(* Logix 5000 project; controller Laser_Cutter vendor 1 type 14 code 149 rev 28.11; software revision 28.00 *)

TASK MainTask (continuous, watchdog 500 ms) : MainProgram

MODULES
   Local : vendor 1 type 14 code 149 (Compact 0, rev 28.11)
      DI1 : 1769-IQ16 (Compact 2, rev 1.1, Input RPI 20 ms)
      Discrete_IO : Embedded (Compact 1, rev 3.1, Output RPI 20 ms)
      ASCII_Comms_Modual : vendor 1 type 109 code 66 (Compact 3, rev 2.1, Output RPI 2 ms)   // Modual for serial communication with the laser controller
      MURR_IMPACT_IO_1 : vendor 640 type 7 code 55085 (Ethernet 192.168.1.40, rev 1.1, StandardDataDriven RPI 20 ms)
      MURR_IMPACT_IO_2 : vendor 640 type 7 code 55085 (Ethernet 192.168.1.41, rev 1.1, StandardDataDriven RPI 20 ms)
END_MODULES

TYPE CON_EIP_IN :
STRUCT
   targetPosition : DINT;
   positioningBand : DINT;
   speed : DINT;
   zoneBoundaryPos : DINT;
   zoneBoundaryNeg : DINT;
   acceleration : INT;
   deceleration : INT;
   pressingCurrentLimit : INT;
   loadCurrentThreshold : INT;
   cs1_UNAVAILABLE_0 : BOOL;
   PUSH : BOOL;
   DIR : BOOL;
   INC : BOOL;
   GSL0 : BOOL;
   GSL1 : BOOL;
   MOD0 : BOOL;
   MOD1 : BOOL;
   ASO0 : BOOL;
   ASO1 : BOOL;
   SMOD : BOOL;
   cs1_UNAVAILABLE_11 : BOOL;
   NTC0 : BOOL;
   NTC1 : BOOL;
   cs1_UNAVAILABLE_14 : BOOL;
   cs1_UNAVAILABLE_15 : BOOL;
   DSTR : BOOL;
   HOME : BOOL;
   STP : BOOL;
   RES : BOOL;
   SON : BOOL;
   JISL : BOOL;
   JVEL : BOOL;
   JOG_NEG : BOOL;
   JOG_POS : BOOL;
   cs2_UNAVAILABLE_9 : BOOL;
   cs2_UNAVAILABLE_10 : BOOL;
   cs2_UNAVAILABLE_11 : BOOL;
   cs2_UNAVAILABLE_12 : BOOL;
   cs2_UNAVAILABLE_13 : BOOL;
   RMOD : BOOL;
   BKRL : BOOL;
END_STRUCT
END_TYPE

TYPE CON_EIP_OUT :
STRUCT
   currentPosition : DINT;
   commandCurrent : DINT;
   currentSpeed : DINT;
   alarmCode : INT;
   UNAVAILABLE_14 : SINT;
   UNAVAILABLE_15 : SINT;
   UNAVAILABLE_16 : SINT;
   UNAVAILABLE_17 : SINT;
   UNAVAILABLE_18 : SINT;
   UNAVAILABLE_19 : SINT;
   totalMovingCount : DINT;
   totalMovingDistance : DINT;
   ALML : BOOL;
   ss1_UNAVAILABLE_1 : BOOL;
   ss1_UNAVAILABLE_2 : BOOL;
   ss1_UNAVAILABLE_3 : BOOL;
   ss1_UNAVAILABLE_4 : BOOL;
   ss1_UNAVAILABLE_5 : BOOL;
   ss1_UNAVAILABLE_6 : BOOL;
   ss1_UNAVAILABLE_7 : BOOL;
   ss1_UNAVAILABLE_8 : BOOL;
   ss1_UNAVAILABLE_9 : BOOL;
   ss1_UNAVAILABLE_10 : BOOL;
   ss1_UNAVAILABLE_11 : BOOL;
   ss1_UNAVAILABLE_12 : BOOL;
   ss1_UNAVAILABLE_13 : BOOL;
   ss1_UNAVAILABLE_14 : BOOL;
   ss1_UNAVAILABLE_15 : BOOL;
   PEND : BOOL;
   HEND : BOOL;
   MOVE : BOOL;
   ALM : BOOL;
   SV : BOOL;
   PSFL : BOOL;
   PUSH : BOOL;
   GHMS : BOOL;
   RMDS : BOOL;
   TRQS : BOOL;
   LOAD : BOOL;
   PZONE : BOOL;
   ZONE1 : BOOL;
   ZONE2 : BOOL;
   PWR : BOOL;
   EMGS : BOOL;
END_STRUCT
END_TYPE

TYPE POSITIONS :
STRUCT
   POSITIONS : DINT;
END_STRUCT
END_TYPE

TYPE savedRecipes :   // Array of Saved Recipes from HMI
STRUCT
   programOrder : DINT[20];
   numberOfSteps : DINT;
   numZonesBeforeNextStep : DINT[20];
   numXZones : DINT;
   numYZones : DINT;
   recipeName : STRING;
END_STRUCT
END_TYPE

TYPE savedRecipes111 :   // Array of Recipes Saved from HMI
STRUCT
   A : DINT[20];
   B : DINT[20];
   C : DINT[20];
   D : DINT[20];
   E : DINT[20];
   F : DINT[20];
   G : DINT[20];
   H : DINT[20];
   I : DINT[20];
   J : DINT[20];
   K : DINT[20];
   L : DINT[20];
   M : DINT[20];
   N : DINT[20];
   O : DINT[20];
   P : DINT[20];
   Q : DINT[20];
   R : DINT[20];
   S : DINT[20];
   T : DINT[20];
END_STRUCT
END_TYPE

ADD_ON_INSTRUCTION Value_Within_Tolerance   (* revision 1.0 *)
VAR_OUTPUT
   Within_Tolerance : BOOL; {access Read Only, visible}
END_VAR
VAR_INPUT
   Process_Value : DINT; {required}
   Setpoint_Value : DINT; {required}
   Tolerance : DINT; {required}
END_VAR
VAR
   Hi_Limit : DINT; {access None}
   Lo_Limit : DINT; {access None}
END_VAR

ROUTINE Logic   (* ladder *)
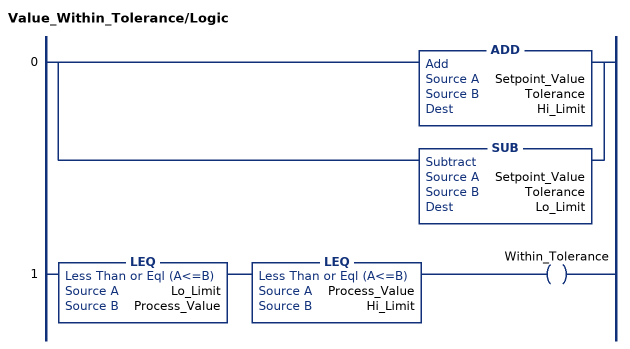
   0: [ADD(Setpoint_Value,Tolerance,Hi_Limit) ,SUB(Setpoint_Value,Tolerance,Lo_Limit) ];
   1: LEQ(Lo_Limit,Process_Value)LEQ(Process_Value,Hi_Limit)OTE(Within_Tolerance);
END_ROUTINE
END_ADD_ON_INSTRUCTION

VAR_GLOBAL   (* controller tags *)
   alarmResetPB : BOOL;   // Global Alarm Reset PB
   audibleAlarm : ALIAS FOR Local:1:O.Data.3;
   bearingConveyorDriveAlarm : ALIAS FOR Local:1:I.Data.6;
   blowOffOn : ALIAS FOR Local:1:O.Data.9;
   boltDriverDown : ALIAS FOR MURR_IMPACT_IO_1:I.Data[1].6;
   boltDriverUp : ALIAS FOR MURR_IMPACT_IO_1:I.Data[1].5;
   boltFeedingBowlOn : ALIAS FOR Local:1:O.Data.7;
   boltFeedingTrackHighLevel : ALIAS FOR MURR_IMPACT_IO_1:I.Data[0].3;
   boltFeedingTrackLowLevel : ALIAS FOR MURR_IMPACT_IO_1:I.Data[0].2;
   boltFeedingTrackOn : ALIAS FOR Local:1:O.Data.8;
   boltPresentAtInfeed : ALIAS FOR MURR_IMPACT_IO_1:I.Data[0].5;
   cameraBadPart : ALIAS FOR Local:1:I.Data.8;
   cameraGoodPart : ALIAS FOR Local:1:I.Data.7;
   cameraOnline : ALIAS FOR Local:1:I.Data.9;
   cameraTrigger : ALIAS FOR Local:1:O.Data.11;
   clampStation2 : ALIAS FOR MURR_IMPACT_IO_1:I.Data[1].7;
   clampStation4 : ALIAS FOR MURR_IMPACT_IO_1:I.Data[2].1;
   clampStation5 : ALIAS FOR MURR_IMPACT_IO_1:I.Data[2].3;
   collarAtStation1 : ALIAS FOR MURR_IMPACT_IO_1:I.Data[0].6;
   collarAtStation2 : ALIAS FOR MURR_IMPACT_IO_1:I.Data[0].7;
   collarAtStation3 : ALIAS FOR MURR_IMPACT_IO_1:I.Data[1].0;
   collarAtStation4 : ALIAS FOR MURR_IMPACT_IO_1:I.Data[1].1;
   collarAtStation5 : ALIAS FOR MURR_IMPACT_IO_1:I.Data[1].2;
   collarFeedingBowlOn : ALIAS FOR Local:1:O.Data.5;
   collarFeedingTrackHighLevel : ALIAS FOR MURR_IMPACT_IO_1:I.Data[0].1;
   collarFeedingTrackLowLevel : ALIAS FOR MURR_IMPACT_IO_1:I.Data[0].0;
   collarFeedingTrackOn : ALIAS FOR Local:1:O.Data.6;
   collarPresentAtInfeed : ALIAS FOR MURR_IMPACT_IO_1:I.Data[0].4;
   currentUser : DINT := 4;   // Access Level of current user
   cycleStartPB : ALIAS FOR Local:1:I.Data.3;
   doorLocksControlRelay : ALIAS FOR Local:1:O.Data.4;
   doorOpenedSafetyRelayStatus : ALIAS FOR Local:1:I.Data.1;
   doorSafetySwitchUnlockSol : ALIAS FOR Local:1:O.Data.10;
   engArrayFullFault : BOOL;
   ESTOP_PB : BOOL;
   eStopSafetyRelayStatus : ALIAS FOR Local:1:I.Data.0;
   greenStatusLight : ALIAS FOR Local:1:O.Data.2;
   keyResetRequired : BOOL;
   leadArrayFullFault : BOOL;
   Local1IData10 : ALIAS FOR Local:1:I.Data.10;
   Local1IData11 : ALIAS FOR Local:1:I.Data.11;
   Local1IData12 : ALIAS FOR Local:1:I.Data.12;
   Local1IData13 : ALIAS FOR Local:1:I.Data.13;
   Local1IData14 : ALIAS FOR Local:1:I.Data.14;
   Local1IData15 : ALIAS FOR Local:1:I.Data.15;
   Local2OData12 : ALIAS FOR Local:1:O.Data.12;
   Local2OData13 : ALIAS FOR Local:1:O.Data.13;
   Local2OData14 : ALIAS FOR Local:1:O.Data.14;
   Local2OData15 : ALIAS FOR Local:1:O.Data.15;
   mainAirOk : ALIAS FOR Local:1:I.Data.2;
   operArrayFullFault : BOOL;
   redStatusLight : ALIAS FOR Local:1:O.Data.0;
   rejectShuttleAtAccept : ALIAS FOR MURR_IMPACT_IO_1:I.Data[2].5;
   rejectShuttleAtReject : ALIAS FOR MURR_IMPACT_IO_1:I.Data[2].6;
   resetPB : ALIAS FOR Local:1:I.Data.5;
   stopPB : ALIAS FOR Local:1:I.Data.4;
   supArrayFullFault : BOOL;
   tapDown : ALIAS FOR MURR_IMPACT_IO_1:I.Data[1].4;
   tapForward : ALIAS FOR MURR_IMPACT_IO_2:O.Data[0].0;
   tapReverse : ALIAS FOR MURR_IMPACT_IO_2:O.Data[0].1;
   tapUp : ALIAS FOR MURR_IMPACT_IO_1:I.Data[1].3;
   TO_DRV1 : CON_EIP_IN := (targetPosition := 12411, positioningBand := 10, speed := 14288, acceleration := 30, deceleration := 30);
   TO_DRV2 : CON_EIP_IN := (targetPosition := 20010, positioningBand := 100, speed := 14288, acceleration := 30, deceleration := 30);
   unclampStation2 : ALIAS FOR MURR_IMPACT_IO_1:I.Data[2].0;
   unclampStation4 : ALIAS FOR MURR_IMPACT_IO_1:I.Data[2].2;
   unclampStation5 : ALIAS FOR MURR_IMPACT_IO_1:I.Data[2].4;
   walkingBeamDown : ALIAS FOR MURR_IMPACT_IO_2:I.Data[0].0;
   walkingBeamLeft : ALIAS FOR MURR_IMPACT_IO_2:I.Data[0].2;
   walkingBeamRight : ALIAS FOR MURR_IMPACT_IO_2:I.Data[0].1;
   walkingBeamUp : ALIAS FOR MURR_IMPACT_IO_1:I.Data[2].7;
   yellowStatusLight : ALIAS FOR Local:1:O.Data.1;
END_VAR

PROGRAM MainProgram   (* main routine MainRoutine *)
VAR
   aAcceptPartSol : BOOL;
   aBlowOffOnSol : BOOL;
   aBlowoffTimer : TIMER := (PRE := 1000);
   aBoltBowlFeedingOn : BOOL;
   aBoltDriverDownSol : BOOL;
   aBoltDriverForward : BOOL;
   aBoltDriverReverse : BOOL;
   aBoltDriverUpSol : BOOL;
   aBoltFeedingTrackOn : BOOL;
   aCameraTrigger : BOOL;
   acceptPartSol : BOOL;
   aClampingStation2Down : BOOL;
   aClampingStation2Up : BOOL;
   aClampingStation4DownSol : BOOL;
   aClampingStation5DownSol : BOOL;
   aClampingStation5UpSol : BOOL;
   aCollarBowlFeedingOn : BOOL;
   aCollarFeedingTrackOn : BOOL;
   aDoorSafetySwitchUnlockSol : BOOL;
   aExhaustStart : BOOL := 1;
   airInitDebounceTimer : TIMER := (PRE := 10000);
   airPressureAlarmTimer : TIMER := (PRE := 4000);
   alarmActive : BOOL;
   alarmActiveOneShot : BOOL;
   alarmActiveOneShotStorage : BOOL;
   alarmMessageBuffer : STRING;
   alarmResetPressed : BOOL;
   alarmResetPressedTmr : TIMER := (PRE := 1000);
   alarmString1 : STRING[35] := ([0] := 'Estop Pressed During Initialization', [1] := 'Door Not Locked During Initialization', [2] := 'Low Air Presure During Initialization', [3] := 'Front Pallet Shotpin Failed to Extend During Initialitzation', [4] := 'Back Pallet Shotpin Failed to Extend During Initialitzation', [5] := 'Estop Pressed During Cycle', [6] := 'Door Opened During Cycle', [7] := 'No Main Air Presure During Cycle', [8] := 'Front Pallet Shotpin Failed to Extend During Cycle', [9] := 'Front Pallet Shotpin Failed to Retract During Cycle', [10] := 'Back Pallet Shotpin Failed to Extend During Cycle', [11] := 'Back Pallet Shotpin Failed to Retract During Cycle', [12] := 'Laser Error', [13] := 'X Axis Failed to Move Home', [14] := 'X Axis Failed to Move to Load', [15] := 'X Axis Failed to Move to Current Zone', [16] := 'X Axis Servo Drive Alarm', [17] := 'X Axis Drive Failed to Enable', [18] := 'X Axis Drive Failed to Disable', [19] := 'Y Axis Failed to Move Home', [20] := 'Y Axis Failed to Move to Load', [21] := 'Y Axis Failed to Move to Current Zone', [22] := 'Y Axis Servo Drive Alarm', [23] := 'Y Axis Drive Failed to Enable', [24] := 'Y Axis Drive Failed to Disable', [25] := 'Laser Timeout Error', [26] := 'External Laser Shutter Failure to Close During Initialization', [27] := 'External Laser Shutter Failure to Close During Cycle', [28] := 'External Laser Shutter Failure to Open During Cycle', [29] := 'Exhaust Arm Not In Position', [30] := 'Low Exhaust Air Flow', [31] := 'User Level Array Full', [32] := 'Low Air Pressure During Cycle', [33] := 'MANUAL MODE ACTIVATED DURING CYCLE');
   alarmString2 : STRING[32];
   alarmStringBuffer : STRING;
   alarmTmr1 : TIMER[32] := ([0].PRE := 100000, [1].PRE := 10000, [2].PRE := 3000, [3].PRE := 3000, [4].PRE := 3000, [5].PRE := 500, [6].PRE := 20000, [7].PRE := 10000, [8].PRE := 10000, [9].PRE := 5000, [10].PRE := 20000, [11].PRE := 10000, [12].PRE := 10000, [13].PRE := 3000, [14].PRE := 20000, [15].PRE := 10000, [16].PRE := 10000, [17].PRE := 3000, [18].PRE := 20000, [19].PRE := 40000, [20].PRE := 10000, [21].PRE := 3000, [22].PRE := 3000, [24].PRE := 500, [25].PRE := 3000, [26].PRE := 3000, [27].PRE := 3000, [28].PRE := 3000, [30].PRE := 3000, [31].PRE := 3000);
   alarmTmr2 : TIMER[32] := ([0].PRE := 3000, [1].PRE := 3000, [2].PRE := 3000, [3].PRE := 3000, [4].PRE := 8000, [5].PRE := 500, [6].PRE := 5000, [7].PRE := 3000, [10].PRE := 3000, [11].PRE := 3000, [13].PRE := 3000, [14].PRE := 3000, [15].PRE := 3000, [17].PRE := 3000, [18].PRE := 3000, [20].PRE := 3000, [21].PRE := 3000, [22].PRE := 3000, [24].PRE := 3000, [25].PRE := 3000, [27].PRE := 3000, [28].PRE := 3000, [30].PRE := 3000);
   aRejectPartSol : BOOL;
   aTapForward : BOOL;
   aTapReverse : BOOL;
   automaticSeqStep : DINT;
   autoMode : BOOL := 1;
   autoModeReady : BOOL := 1;
   aWalkingBeamDownSol : BOOL;
   aWalkingBeamLeftSol : BOOL;
   aWalkingBeamRightSol : BOOL;
   aWalkingBeamUpSol : BOOL;
   blowoffSeqStep : DINT;
   boltBowlFeedingOn : BOOL;
   boltDriverDownDB : TIMER := (PRE := 50);
   boltDriverDownSol : BOOL;
   boltDriverForward : BOOL;
   boltDriverReverse : BOOL;
   boltDriverSeqStep : DINT;
   boltDriverToStartPOS : BOOL;
   boltDriverToStartPOSdb : TIMER := (PRE := 400);
   boltDriverUpDB : TIMER := (PRE := 50);
   boltDriverUpSol : BOOL;
   boltPresentAtInfeedDB : TIMER := (PRE := 50);
   calcZonesDone : BOOL;
   cameraTriggerFlag : BOOL;
   cameraTriggerPulse : TIMER := (PRE := 500);
   clampingStation2Down : BOOL;
   clampingStation2Up : BOOL;
   clampingStation4DownSol : BOOL;
   clampingStation4UpSol : BOOL;
   clampingStation5DownSol : BOOL;
   clampingStation5Sol : BOOL;
   clampStation2DB : TIMER := (PRE := 50);
   clampStation4DB : TIMER := (PRE := 50);
   clampStation5DB : TIMER := (PRE := 50);
   collarAtStation1DB : TIMER := (PRE := 50);
   collarAtStation2DB : TIMER := (PRE := 50);
   collarAtStation3DB : TIMER := (PRE := 50);
   collarAtStation4DB : TIMER := (PRE := 50);
   collarAtStation5DB : TIMER := (PRE := 50);
   collarBowlFeedingOn : BOOL;
   collarFeedingTrackHighLevelDB : TIMER := (PRE := 50);
   collarFeedingTrackLowLevelDB : TIMER := (PRE := 50);
   collarPresentAtInfeedDB : TIMER := (PRE := 50);
   Counter : DINT;
   Counter2 : DINT;
   Counter3 : DINT;
   CYCLE_ALM : DINT;
        .4   // Front Shotpin Failed to Retract During Cycle
        .2   // No Main Air Pressure During Cycle Alarm
        .3   // Front Shotpin Failed to Extend During Cycle
        .1   // Door Opened During Cycle Alarm
        .6   // Back Shotpin Failed to Retract During Cycle
        .5   // Back Shotpin Failed to Extend During Cycle
        .0   // EStop Pressed During Cycle Alarm
        .7   // Laser Error
   CYCLE_ALM_TMR : TIMER[15] := ([3].PRE := 3000, [4].PRE := 3000, [5].PRE := 3000, [6].PRE := 3000, [7].PRE := 3000, [8].PRE := 3000, [9].PRE := 10000, [10].PRE := 250);
   CYCLE_COMPLETE : BOOL;
   CYCLE_IN_PROG : BOOL;
   cycleComplete : BOOL;
   cycleInProgDebounce : TIMER := (PRE := 15000);
   cycleTimeBufferMin : DINT;
   cycleTimeBufferSec : DINT := 2;
   cycleTimer : TIMER := (PRE := 99999999, ACC := 78863958, EN := 1, TT := 1);
   cycleTimerBuffer : DINT;
   doorClosedDebounceTimer : TIMER := (PRE := 50, ACC := 50, EN := 1, DN := 1);
   doorLockAtInitialPosition : BOOL := 1;
   doorLockedDebounceTimer : TIMER := (PRE := 50, ACC := 50, EN := 1, DN := 1);
   doorUnlockedDebounceTimer : TIMER := (PRE := 50);
   empty_string : STRING;
   exeBlowoffSR : BOOL;
   Exec_Bolt_Driver_SR : BOOL;
   Exec_Drive_Bolt : BOOL;
   Exec_Laser_SR : BOOL;
   Exec_Robot_SR : BOOL;
   Exec_Tapping_SR : BOOL;
   execLoadPalletSR : BOOL;
   Execute_BlowoffSR : BOOL;
   Execute_MoveToZoneSR : BOOL;
   Execute_RejectSR : BOOL;
   Execute_VisionInspectionSR : BOOL;
   executeInitializationSequence : BOOL;
   exeCycleStationsSR : BOOL;
   exeInfeedBoltSR : BOOL;
   exeInfeedCollarSR : BOOL;
   exeInspectionSR : BOOL;
   exeRobotSR : BOOL;
   exeScrewBoltSR : BOOL;
   exeTappingSR : BOOL;
   HAND_GREEN_STATUS_LIGHT : BOOL;
   HAND_RED_STATUS_LIGHT : BOOL;
   HAND_YELLOW_STATUS_LIGHT : BOOL;
   HMI_AutoMode_Req : BOOL;
   HMI_ManualMode_Req : BOOL;
   HMI_MESSAGE_NUM : DINT := 16;
   hmiMessageNumber : DINT := 16;
   hmiMessageNumberBuffer : DINT := 16;
   hmiMessageString : STRING := 'READY TO BEGIN CYCLE';
   hmiMessageStringArray : STRING[64] := ([1] := 'ALARM ACTIVE$0D$0APRESS RESET FAULT BUTTON', [2] := 'OFF MODE', [3] := 'MANUAL MODE ACTIVE', [4] := 'EMERGENCY STOP BUTTON PRESSED', [5] := 'RESET OF ESTOP REQUIRED - PUSH RESET BUTTON', [6] := 'SYSTEM INITIALIZATION REQUIRED', [7] := 'INITIALIZATION IN PROGRESS', [8] := 'LASER ERROR - RESET LASER BY TURNING KEY SWITCH OFF AND ON AGAIN', [9] := 'LASER WARNING ACTIVE', [10] := 'DRIVE 1 REQUIRES HOMING', [11] := 'DRIVE 2 REQUIRES HOMING', [12] := 'PALLET NOT PRESENT', [13] := 'CLOSE DOOR AND PRESS POWER ON TO RESET', [14] := 'CYCLE COMPLETE$0D$0AREMOVE PALLET', [15] := 'READY TO LOAD NEW PALLET', [16] := 'READY TO BEGIN CYCLE', [17] := 'AUTOMATIC RUN IN PROGRESS', [18] := 'TEST IN PROGRESS$0D$0APLEASE WAIT', [21] := 'MOVING TO LOAD POSITION FOR END OF RUN$0D$0APLEASE WAIT', [22] := 'REMOVE INSTRUMENT TO COMPLETE RUN', [23] := 'MOVING TO LOAD POSITION TO REPLACE SULU$0D$0APLEASE WAIT', [24] := 'REMOVE INSTRUMENT AND REPLACE SULU', [25] := 'MOVING TO LOAD POSITION$0D$0APLEASE WAIT', [26] := 'MOVING TO 90 DEG MESH LOADING POSITION$0D$0APLEASE WAIT', [27] := 'MOVING TO 65 DEG MESH LOADING POSITION$0D$0APLEASE WAIT', [28] := 'REPLACE 90 DEG MESH AND$0D$0APRESS THE ACKNOWLEDGE BUTTON TO CONFIRM', [29] := 'REPLACE 65 DEG MESH AND$0D$0APRESS THE ACKNOWLEDGE BUTTON TO CONFIRM', [30] := 'ACTIVATE OPTOTOUCH TO MOVE TO LOADING POSITION', [31] := 'ACTIVATE OPTOTOUCH TO MOVE TO LOADING POSITION$0D$0AAFTER THE ALARM', [32] := 'MOVING TO LOADING POSITION$0D$0AAFTER AN ALARM', [33] := 'INSTALL OR RE-POSITION RELIATACK HANDLE NEST', [34] := 'MOVING TO SHORT ABSTACK MESH LOADING POSITION$0D$0APLEASE WAIT', [35] := 'REPLACE SHORT ABSTACK MESH AND$0D$0APRESS THE ACKNOWLEDGE BUTTON TO CONFIRM', [36] := 'MOVING TO LOAD POSITION TO REPLACE INSTRUMENT$0D$0APLEASE WAIT', [37] := 'REMOVE AND REPLACE INSTRUMENT', [50] := 'PRINTING LAST SAMPLE LABELS$0D$0AFOR LABEL CHECKING', [51] := 'PRESS REPRINT ALL LABELS BUTTON', [52] := 'PRINTING SUMMARY LABELS$0D$0APLEASE WAIT', [53] := 'PRESS REPRINT SUMMARY LABELS BUTTON');
   idleTime : TIMER := (PRE := 99999999, ACC := 48278377, EN := 1, TT := 1);
   idleTimeBuffer : DINT;
   idleTimeBufferMin : DINT := 804;
   idleTimeBufferSec : DINT := 38;
   INIT_ALM : DINT;
        .4   // Back Shotpin Failed to Retract During Initialiazation
        .2   // No Main Air Pressure During Initialization Alarm
        .0   // EStop Pressed During Initialization Alarm
        .1   // Door Failed to Lock Durring Initialiaztion
        .3   // Front Shotpin Failed to Retract During Initialiazation
   INIT_ALM_TMR : TIMER[10] := ([3].PRE := 3000, [4].PRE := 3000, [5].PRE := 3000, [6].PRE := 3000);
   INIT_IN_PROG : BOOL;
   INIT_START_PB : BOOL;
   INIT_START_PB_ONS : BOOL;
   initDelayTimer : TIMER := (PRE := 500);
   initHMIMessageDelayTimer : TIMER := (PRE := 500);
   initializationPushbutton : BOOL;
   InitializationRequired : BOOL;
   Initialize_Timer : TIMER := (PRE := 3000, ACC := 3000, EN := 1, DN := 1);
   initSeqStep : DINT;
   initTimeout : TIMER := (PRE := 10000);
   inspectionSeqStep : DINT;
   lampTestActive : BOOL;
   lampTestPB : BOOL;
   lampTestTimer : TIMER := (PRE := 6000);
   laserMessageSeqStep : INT;
   LaserSeqStep : INT;
   leadingZeros : STRING := '000';
   loadPalletSeqStep : INT;
   mAcceptPartPB : BOOL;
   mAcceptPartSol : BOOL;
   manualMode : BOOL;
   maTapReversePB : BOOL;
   mBlowOffOn : BOOL;
   mBlowOffOnSol : BOOL;
   mBlowOffSol : BOOL;
   mBoltBowlFeedingOnPB : BOOL;
   mBoltDriverDownPB : BOOL;
   mBoltDriverDownSol : BOOL;
   mBoltDriverForward : BOOL;
   mBoltDriverForwardPB : BOOL;
   mBoltDriverReverse : BOOL;
   mBoltDriverReversePB : BOOL;
   mBoltDriverUpPB : BOOL;
   mBoltDriverUpSol : BOOL;
   mBoltFeedingTrackOnPB : BOOL;
   mcameraTrigger : BOOL;
   mClampingStation2Down : BOOL;
   mClampingStation2DownSol : BOOL;
   mClampingStation2Up : BOOL;
   mClampingStation2UpPB : BOOL;
   mClampingStation2UpSol : BOOL;
   mClampingStation4DownSol : BOOL;
   mClampingStation4UpPB : BOOL;
   mClampingStation4UpSol : BOOL;
   mClampingStation5DownPB : BOOL;
   mClampingStation5DownSol : BOOL;
   mClampingStation5UpPB : BOOL;
   mClampingStation5UpSol : BOOL;
   mClampStation4DownPB : BOOL;
   mCollarBowlFeedingOnPB : BOOL;
   mCollarFeedingTrackOnPB : BOOL;
   mDoorSafetySwitchUnlockSol : BOOL;
   MoveToZoneSeqStep : INT;
   mRejectPartPB : BOOL;
   mRejectPartSol : BOOL;
   mSecPulseOffTmr1 : TIMER;
   mSecPulseOnTmr1 : TIMER := (EN := 1, TT := 1);
   mTapForward : BOOL;
   mTapForwardPB : BOOL;
   mTapReverse : BOOL;
   mWalkingBeamDownPB : BOOL;
   mWalkingBeamDownSol : BOOL;
   mWalkingBeamLeftPB : BOOL;
   mWalkingBeamLeftSol : BOOL;
   mWalkingBeamRightPB : BOOL;
   mWalkingBeamRightSol : BOOL;
   mWalkingBeamUpPB : BOOL;
   mWalkingBeamUpSol : BOOL;
   n : TIMER := (PRE := 50);
   noAirDurringCycleAlarmTimer : TIMER := (PRE := 3000);
   nulString : STRING;
   oneSecPulseOffTmr : TIMER := (EN := 1, TT := 1);
   oneSecPulseOnTmr : TIMER;
   p2pCycleTime : TIMER := (PRE := 99999999, ACC := 2605);
   p2pCycleTimeBuffer : DINT := 10001;
   p2pCycleTimeBufferSec : DINT := 10;
   palletpresentDebounceTimer : TIMER := (PRE := 50, ACC := 51, EN := 1, DN := 1);
   palletShotpinExtendedBackDebounceTimer : TIMER := (PRE := 50);
   palletShotpinExtendedFrontDebounceTimer : TIMER := (PRE := 50);
   palletShotpinRetractedDebounceTimer : TIMER := (PRE := 50, ACC := 51, EN := 1, DN := 1);
   partsPresentDurringInitialization : BOOL;
   pause : BOOL := 1;
   performOpControl : CONTROL := (LEN := 6);
   performOperation : DINT[1];
   readyToMovePallet : BOOL;
   readyToStartCycle : BOOL;
   rejectPartFlag : BOOL;
   rejectPartSol : BOOL;
   rejectPartSR : DINT[1];
   rejectSeqStep : DINT;
   rejectShuttleAtAcceptDB : TIMER := (PRE := 50);
   rejectShuttleAtRejectDB : TIMER := (PRE := 50);
   remotePVDisplayNum : DINT;
   resetPartCountingValuesHMIPB : BOOL;
   resetPartCountingValuesTimer : TIMER := (PRE := 3000);
   robotAtDropAPR : BOOL;
   robotAtHome : BOOL;
   robotAtPickAPR : BOOL;
   robotFinishedDrop : BOOL;
   robotHasBolt : BOOL;
   robotInMotion : BOOL;
   robotPickBolt : BOOL;
   robotScrewInBolt : BOOL;
   robotSeqStep : DINT;
   runsCompleted : DINT := 100;
   runTime : TIMER := (PRE := 99999999);
   runTimeBuffer : DINT;
   runTimeBufferMin : DINT;
   runTimeBufferSec : DINT;
   sendRobotToDropAPR : BOOL;
   sendRobotToHome : BOOL;
   sendRobotToPick : BOOL;
   serialPortControl : SERIAL_PORT_CONTROL;
   shortDelay : TIMER := (PRE := 50);
   startCycleTimer : BOOL := 1;
   startP2PTimer : BOOL := 1;
   startRobotSequence : BOOL;
   startRunTimer : BOOL;
   stationNumber : CONTROL := (LEN := 6, POS := 5);
   systemInInitializedPosition : BOOL := 1;
   tapDownDB : TIMER := (PRE := 50);
   tapDwellTimer : TIMER := (PRE := 250);
   tapSeqStep : DINT := 40;
   tapUpDB : TIMER := (PRE := 50);
   testInProgress : BOOL;
   testLaserInZonePB : BOOL := 1;
   testLaserInZonePBONs : BOOL;
   testToggle : BOOL;
   testToggle2 : BOOL := 1;
   TMR_PULSE_OFF : TIMER := (PRE := 500);
   TMR_PULSE_ON : TIMER := (PRE := 500, ACC := 296, EN := 1, TT := 1);
   unclampStation2DB : TIMER := (PRE := 50);
   unclampStation4DB : TIMER := (PRE := 50);
   unclampStation5DB : TIMER := (PRE := 50);
   walkingBeamDownDB : TIMER := (PRE := 50, ACC := 51);
   walkingBeamDownSol : BOOL;
   walkingBeamLeftDB : TIMER := (PRE := 50);
   walkingBeamLeftSol : BOOL;
   walkingBeamRightDB : TIMER := (PRE := 50, ACC := 51);
   walkingBeamRightSol : BOOL;
   walkingBeamUpDB : TIMER := (PRE := 50);
   walkingBeamUpSol : BOOL;
END_VAR

ROUTINE Alarms   (* ladder *)
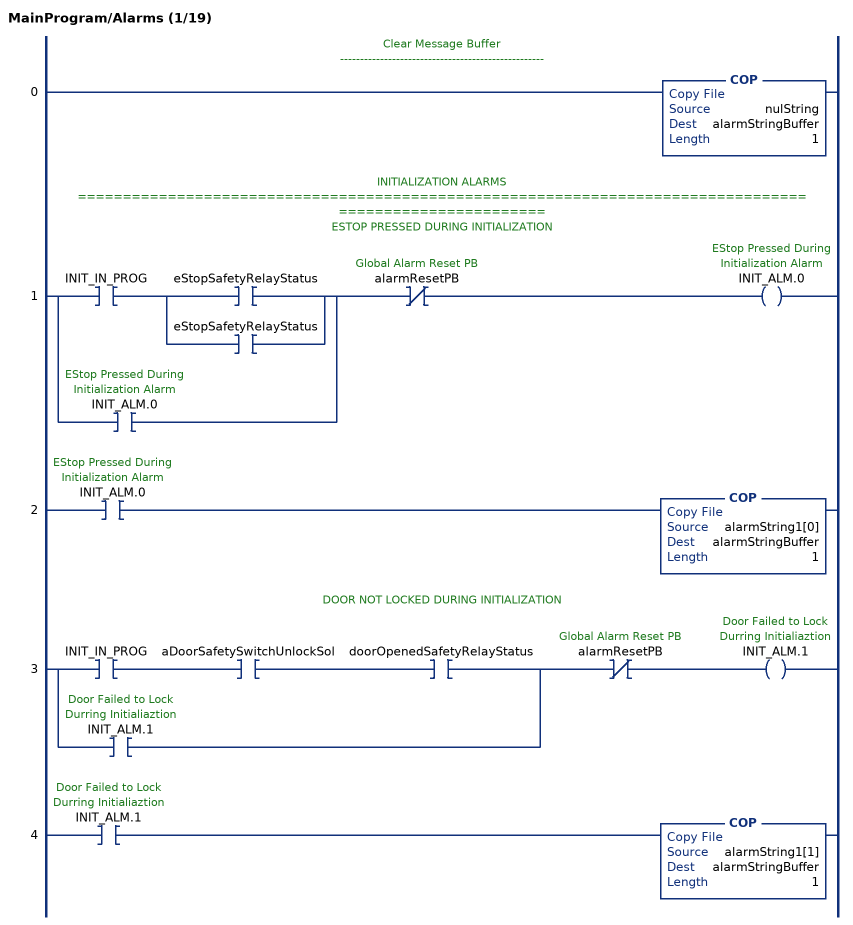
   // Clear Message Buffer
   // ---------------------------------------------------
   0: COP(nulString,alarmStringBuffer,1);
   // INITIALIZATION ALARMS
   // ========================================================================================================
   // ESTOP PRESSED DURING INITIALIZATION
   1: [XIC(INIT_IN_PROG) [XIC(eStopSafetyRelayStatus) ,XIC(eStopSafetyRelayStatus) ] ,XIC(INIT_ALM.0) ]XIO(alarmResetPB)OTE(INIT_ALM.0);
   2: XIC(INIT_ALM.0)COP(alarmString1[0],alarmStringBuffer,1);
   // DOOR NOT LOCKED DURING INITIALIZATION
   3: [XIC(INIT_IN_PROG) XIC(aDoorSafetySwitchUnlockSol) XIC(doorOpenedSafetyRelayStatus) ,XIC(INIT_ALM.1) ]XIO(alarmResetPB)OTE(INIT_ALM.1);
   4: XIC(INIT_ALM.1)COP(alarmString1[1],alarmStringBuffer,1);
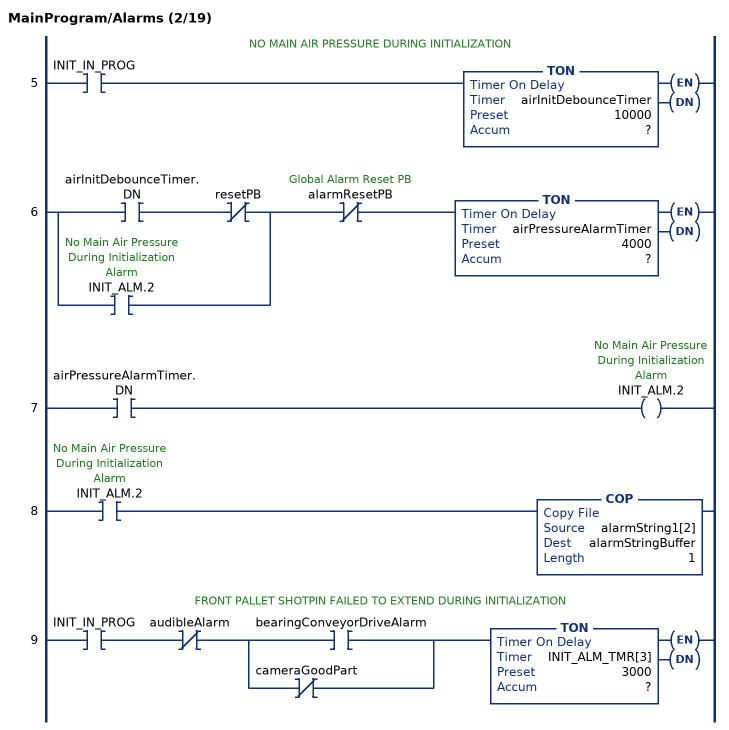
   // NO MAIN AIR PRESSURE DURING INITIALIZATION
   5: XIC(INIT_IN_PROG)TON(airInitDebounceTimer,?,?);
   6: [XIC(airInitDebounceTimer.DN) XIO(resetPB) ,XIC(INIT_ALM.2) ]XIO(alarmResetPB)TON(airPressureAlarmTimer,?,?);
   7: XIC(airPressureAlarmTimer.DN)OTE(INIT_ALM.2);
   8: XIC(INIT_ALM.2)COP(alarmString1[2],alarmStringBuffer,1);
   // FRONT PALLET SHOTPIN FAILED TO EXTEND DURING INITIALIZATION
   9: XIC(INIT_IN_PROG)XIO(audibleAlarm)[XIC(bearingConveyorDriveAlarm) ,XIO(cameraGoodPart) ]TON(INIT_ALM_TMR[3],?,?);
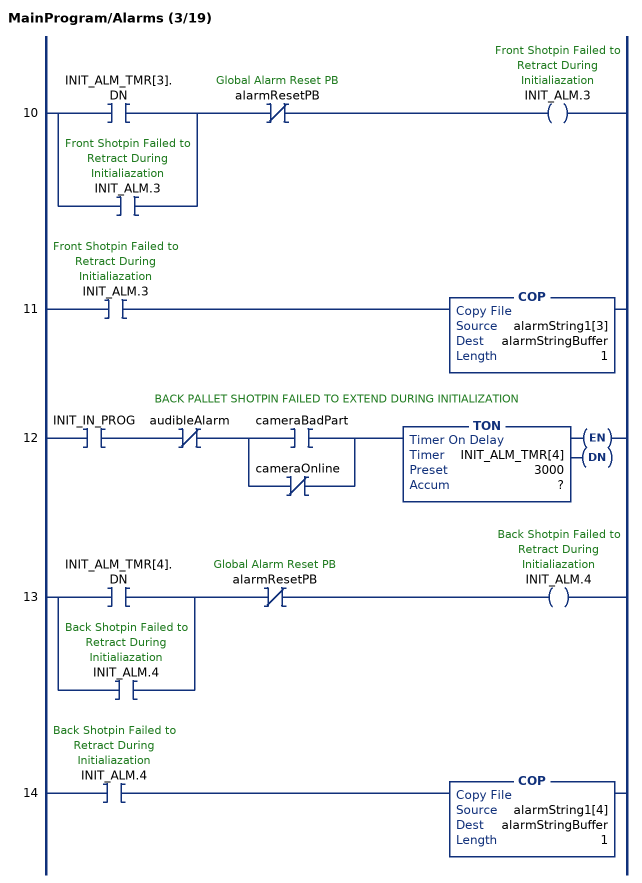
   10: [XIC(INIT_ALM_TMR[3].DN) ,XIC(INIT_ALM.3) ]XIO(alarmResetPB)OTE(INIT_ALM.3);
   11: XIC(INIT_ALM.3)COP(alarmString1[3],alarmStringBuffer,1);
   // BACK PALLET SHOTPIN FAILED TO EXTEND DURING INITIALIZATION
   12: XIC(INIT_IN_PROG)XIO(audibleAlarm)[XIC(cameraBadPart) ,XIO(cameraOnline) ]TON(INIT_ALM_TMR[4],?,?);
   13: [XIC(INIT_ALM_TMR[4].DN) ,XIC(INIT_ALM.4) ]XIO(alarmResetPB)OTE(INIT_ALM.4);
   14: XIC(INIT_ALM.4)COP(alarmString1[4],alarmStringBuffer,1);
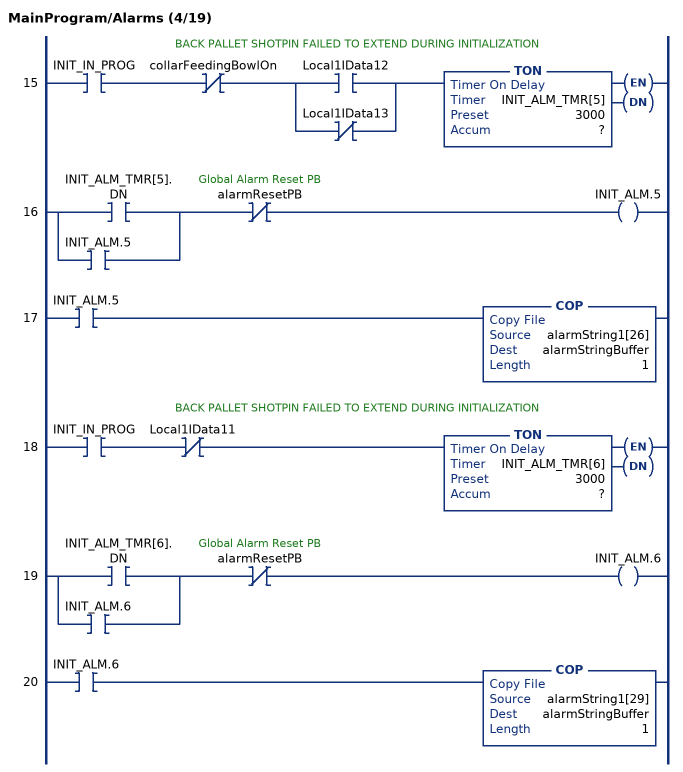
   // BACK PALLET SHOTPIN FAILED TO EXTEND DURING INITIALIZATION
   15: XIC(INIT_IN_PROG)XIO(collarFeedingBowlOn)[XIC(Local1IData12) ,XIO(Local1IData13) ]TON(INIT_ALM_TMR[5],?,?);
   16: [XIC(INIT_ALM_TMR[5].DN) ,XIC(INIT_ALM.5) ]XIO(alarmResetPB)OTE(INIT_ALM.5);
   17: XIC(INIT_ALM.5)COP(alarmString1[26],alarmStringBuffer,1);
   // BACK PALLET SHOTPIN FAILED TO EXTEND DURING INITIALIZATION
   18: XIC(INIT_IN_PROG)XIO(Local1IData11)TON(INIT_ALM_TMR[6],?,?);
   19: [XIC(INIT_ALM_TMR[6].DN) ,XIC(INIT_ALM.6) ]XIO(alarmResetPB)OTE(INIT_ALM.6);
   20: XIC(INIT_ALM.6)COP(alarmString1[29],alarmStringBuffer,1);
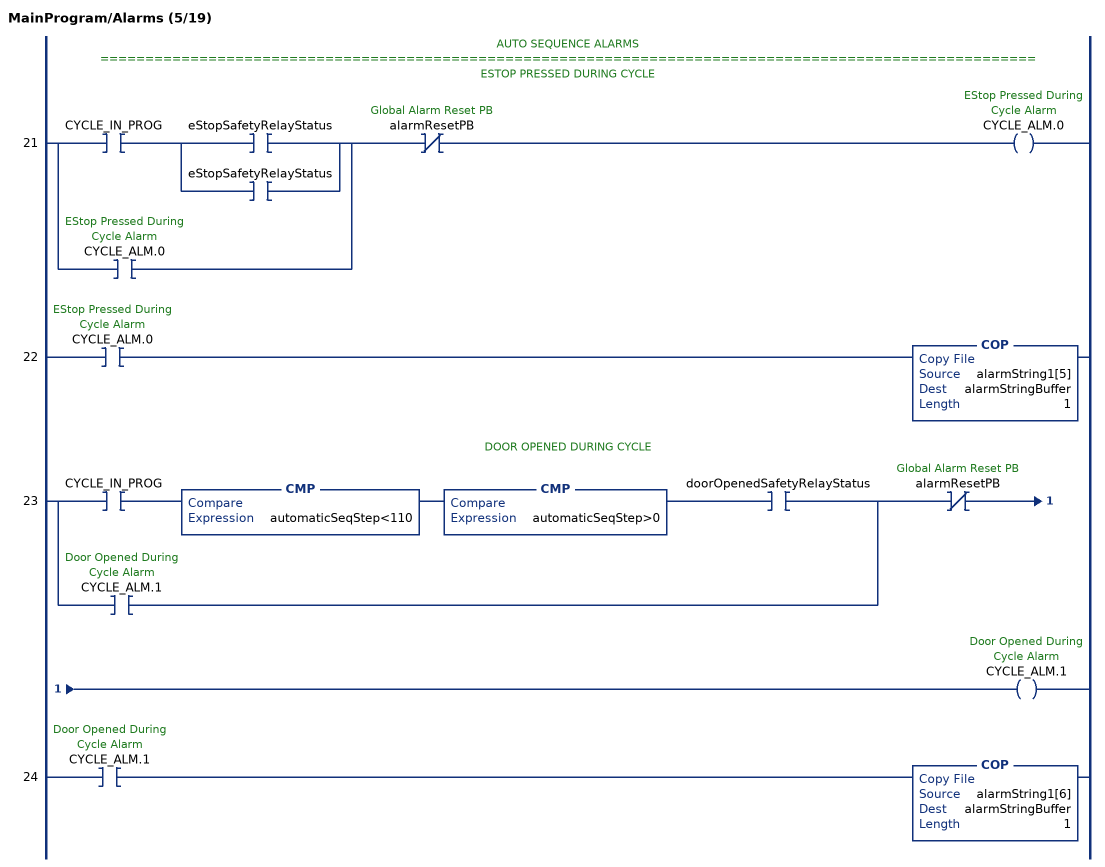
   // AUTO SEQUENCE ALARMS
   // ========================================================================================================
   // ESTOP PRESSED DURING CYCLE
   21: [XIC(CYCLE_IN_PROG) [XIC(eStopSafetyRelayStatus) ,XIC(eStopSafetyRelayStatus) ] ,XIC(CYCLE_ALM.0) ]XIO(alarmResetPB)OTE(CYCLE_ALM.0);
   22: XIC(CYCLE_ALM.0)COP(alarmString1[5],alarmStringBuffer,1);
   // DOOR OPENED DURING CYCLE
   23: [XIC(CYCLE_IN_PROG) CMP(automaticSeqStep<110) CMP(automaticSeqStep>0) XIC(doorOpenedSafetyRelayStatus) ,XIC(CYCLE_ALM.1) ]XIO(alarmResetPB)OTE(CYCLE_ALM.1);
   24: XIC(CYCLE_ALM.1)COP(alarmString1[6],alarmStringBuffer,1);
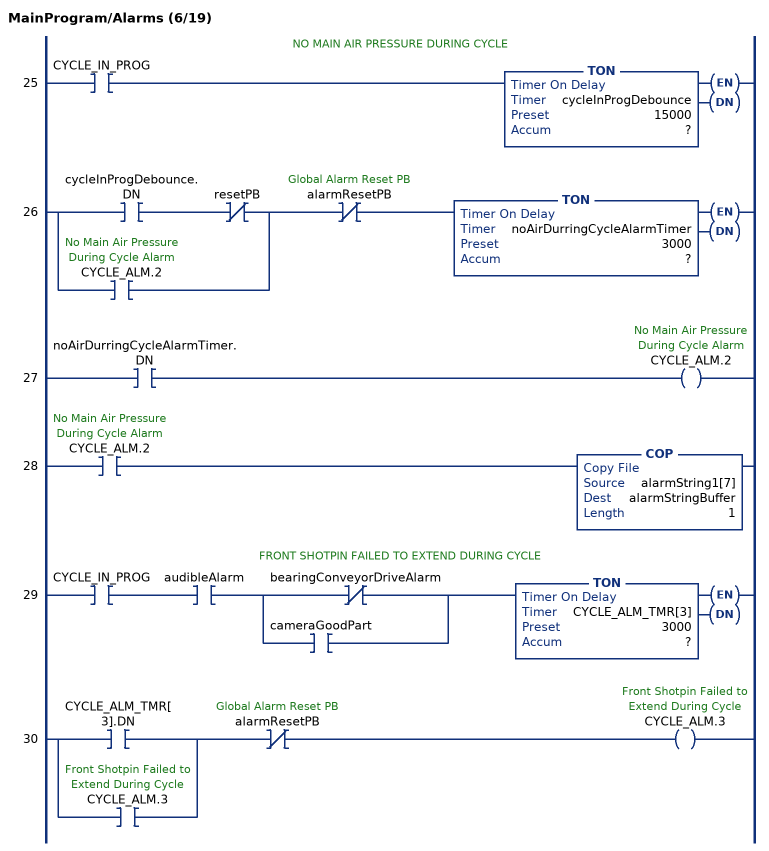
   // NO MAIN AIR PRESSURE DURING CYCLE
   25: XIC(CYCLE_IN_PROG)TON(cycleInProgDebounce,?,?);
   26: [XIC(cycleInProgDebounce.DN) XIO(resetPB) ,XIC(CYCLE_ALM.2) ]XIO(alarmResetPB)TON(noAirDurringCycleAlarmTimer,?,?);
   27: XIC(noAirDurringCycleAlarmTimer.DN)OTE(CYCLE_ALM.2);
   28: XIC(CYCLE_ALM.2)COP(alarmString1[7],alarmStringBuffer,1);
   // FRONT SHOTPIN FAILED TO EXTEND DURING CYCLE
   29: XIC(CYCLE_IN_PROG)XIC(audibleAlarm)[XIO(bearingConveyorDriveAlarm) ,XIC(cameraGoodPart) ]TON(CYCLE_ALM_TMR[3],?,?);
   30: [XIC(CYCLE_ALM_TMR[3].DN) ,XIC(CYCLE_ALM.3) ]XIO(alarmResetPB)OTE(CYCLE_ALM.3);
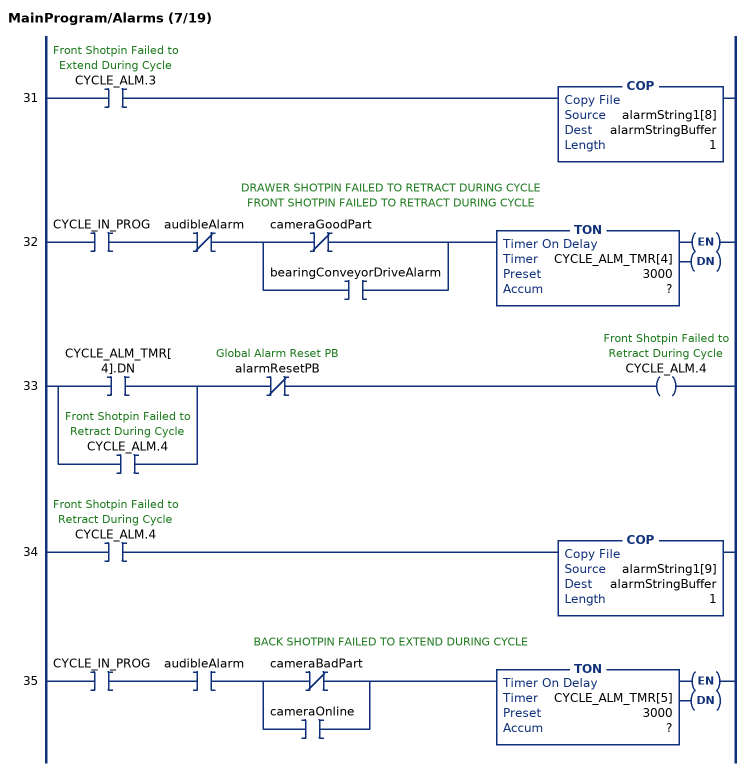
   31: XIC(CYCLE_ALM.3)COP(alarmString1[8],alarmStringBuffer,1);
   // DRAWER SHOTPIN FAILED TO RETRACT DURING CYCLE
   // FRONT SHOTPIN FAILED TO RETRACT DURING CYCLE
   32: XIC(CYCLE_IN_PROG)XIO(audibleAlarm)[XIO(cameraGoodPart) ,XIC(bearingConveyorDriveAlarm) ]TON(CYCLE_ALM_TMR[4],?,?);
   33: [XIC(CYCLE_ALM_TMR[4].DN) ,XIC(CYCLE_ALM.4) ]XIO(alarmResetPB)OTE(CYCLE_ALM.4);
   34: XIC(CYCLE_ALM.4)COP(alarmString1[9],alarmStringBuffer,1);
   // BACK SHOTPIN FAILED TO EXTEND DURING CYCLE
   35: XIC(CYCLE_IN_PROG)XIC(audibleAlarm)[XIO(cameraBadPart) ,XIC(cameraOnline) ]TON(CYCLE_ALM_TMR[5],?,?);
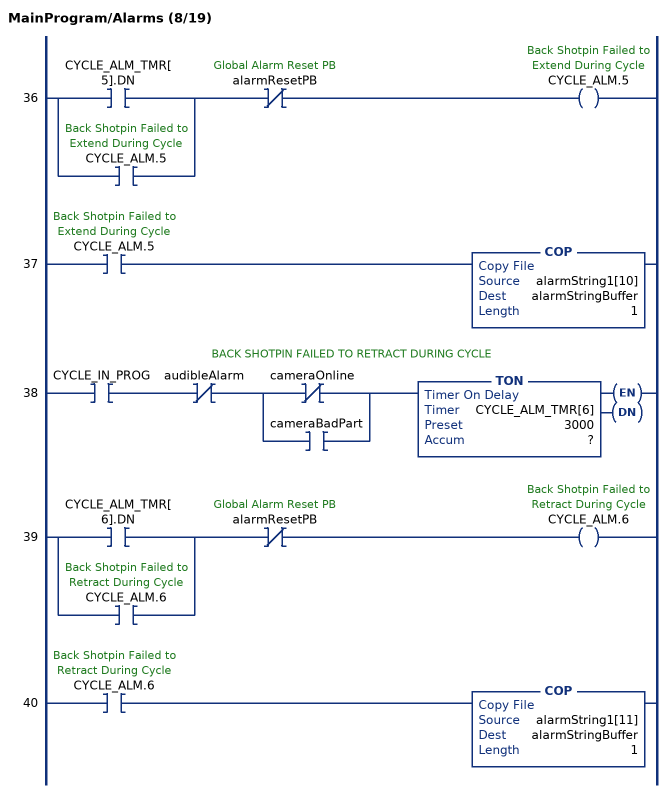
   36: [XIC(CYCLE_ALM_TMR[5].DN) ,XIC(CYCLE_ALM.5) ]XIO(alarmResetPB)OTE(CYCLE_ALM.5);
   37: XIC(CYCLE_ALM.5)COP(alarmString1[10],alarmStringBuffer,1);
   // BACK SHOTPIN FAILED TO RETRACT DURING CYCLE
   38: XIC(CYCLE_IN_PROG)XIO(audibleAlarm)[XIO(cameraOnline) ,XIC(cameraBadPart) ]TON(CYCLE_ALM_TMR[6],?,?);
   39: [XIC(CYCLE_ALM_TMR[6].DN) ,XIC(CYCLE_ALM.6) ]XIO(alarmResetPB)OTE(CYCLE_ALM.6);
   40: XIC(CYCLE_ALM.6)COP(alarmString1[11],alarmStringBuffer,1);
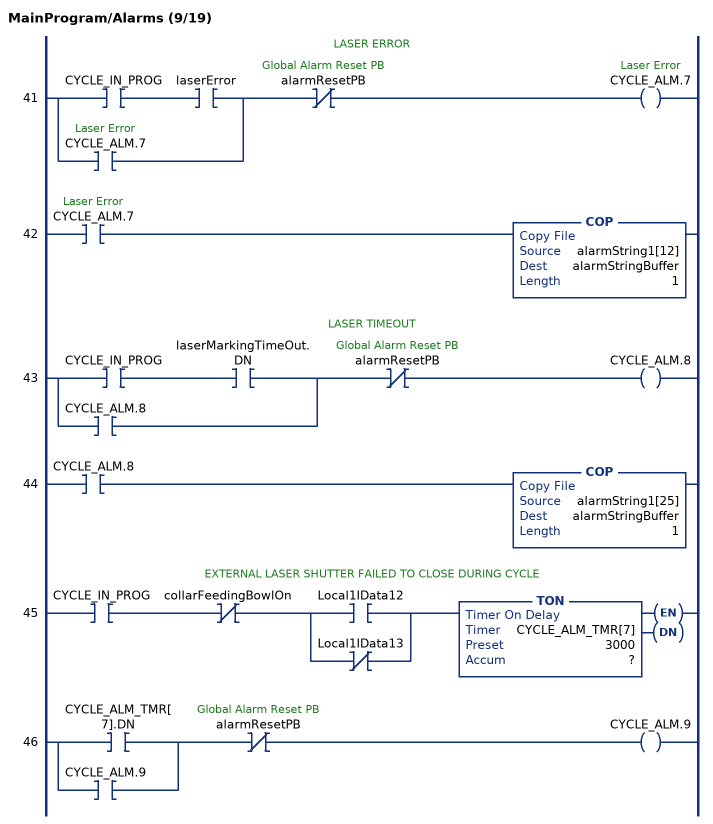
   // LASER ERROR
   41: [XIC(CYCLE_IN_PROG) XIC(laserError) ,XIC(CYCLE_ALM.7) ]XIO(alarmResetPB)OTE(CYCLE_ALM.7);
   42: XIC(CYCLE_ALM.7)COP(alarmString1[12],alarmStringBuffer,1);
   // LASER TIMEOUT
   43: [XIC(CYCLE_IN_PROG) XIC(laserMarkingTimeOut.DN) ,XIC(CYCLE_ALM.8) ]XIO(alarmResetPB)OTE(CYCLE_ALM.8);
   44: XIC(CYCLE_ALM.8)COP(alarmString1[25],alarmStringBuffer,1);
   // EXTERNAL LASER SHUTTER FAILED TO CLOSE DURING CYCLE
   45: XIC(CYCLE_IN_PROG)XIO(collarFeedingBowlOn)[XIC(Local1IData12) ,XIO(Local1IData13) ]TON(CYCLE_ALM_TMR[7],?,?);
   46: [XIC(CYCLE_ALM_TMR[7].DN) ,XIC(CYCLE_ALM.9) ]XIO(alarmResetPB)OTE(CYCLE_ALM.9);
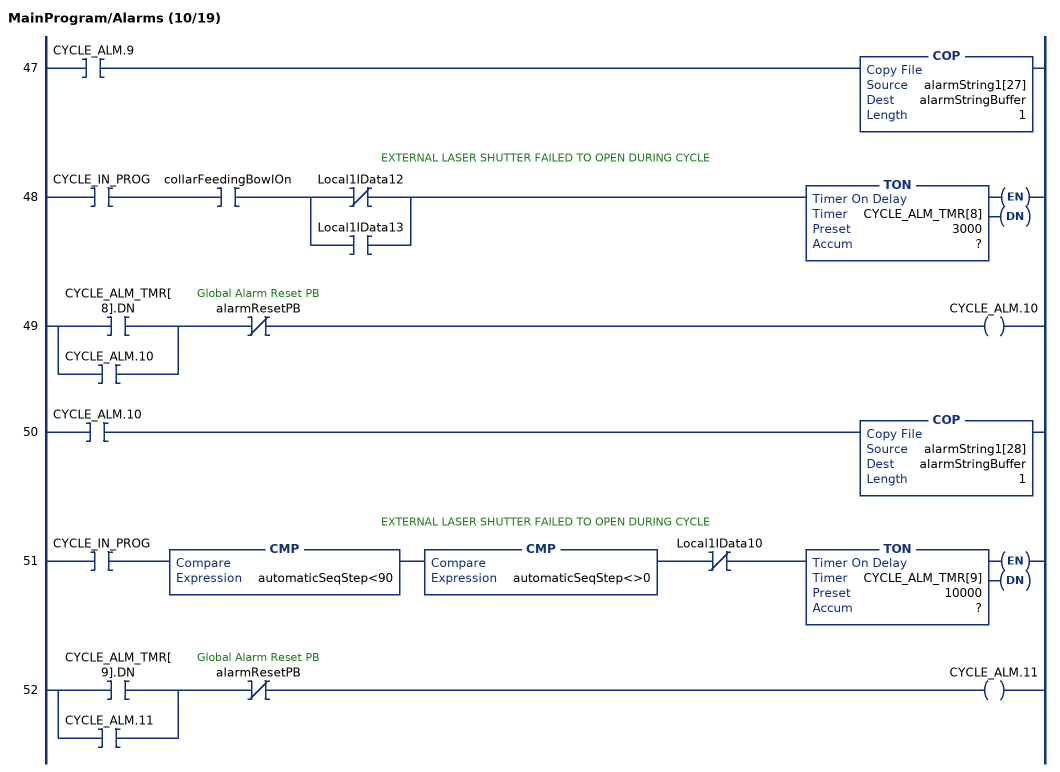
   47: XIC(CYCLE_ALM.9)COP(alarmString1[27],alarmStringBuffer,1);
   // EXTERNAL LASER SHUTTER FAILED TO OPEN DURING CYCLE
   48: XIC(CYCLE_IN_PROG)XIC(collarFeedingBowlOn)[XIO(Local1IData12) ,XIC(Local1IData13) ]TON(CYCLE_ALM_TMR[8],?,?);
   49: [XIC(CYCLE_ALM_TMR[8].DN) ,XIC(CYCLE_ALM.10) ]XIO(alarmResetPB)OTE(CYCLE_ALM.10);
   50: XIC(CYCLE_ALM.10)COP(alarmString1[28],alarmStringBuffer,1);
   // EXTERNAL LASER SHUTTER FAILED TO OPEN DURING CYCLE
   51: XIC(CYCLE_IN_PROG)CMP(automaticSeqStep<90)CMP(automaticSeqStep<>0)XIO(Local1IData10)TON(CYCLE_ALM_TMR[9],?,?);
   52: [XIC(CYCLE_ALM_TMR[9].DN) ,XIC(CYCLE_ALM.11) ]XIO(alarmResetPB)OTE(CYCLE_ALM.11);
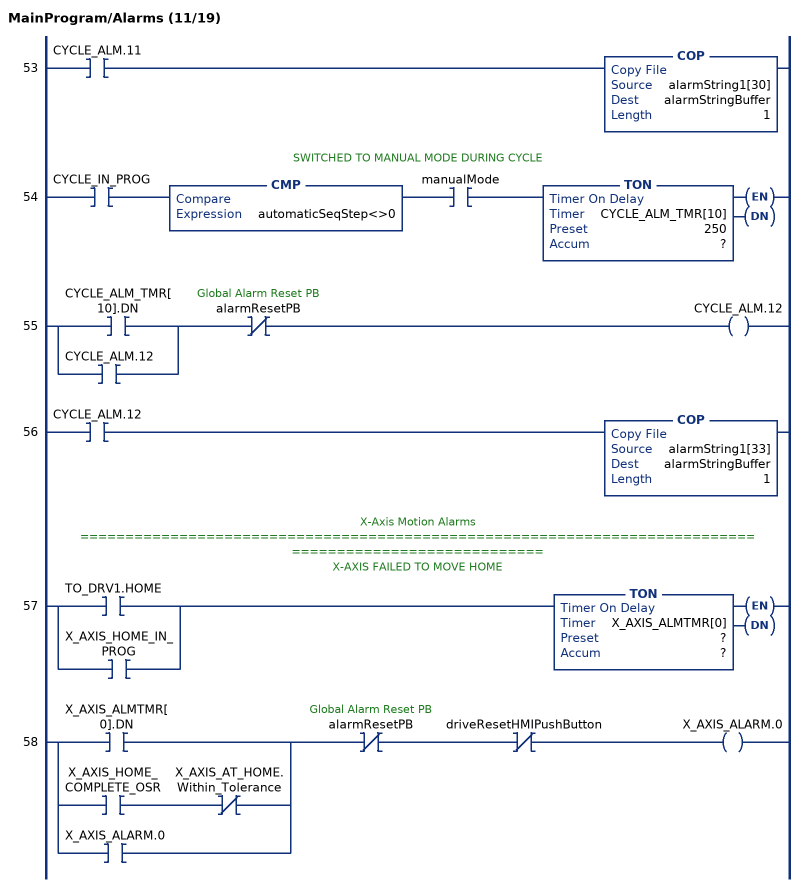
   53: XIC(CYCLE_ALM.11)COP(alarmString1[30],alarmStringBuffer,1);
   // SWITCHED TO MANUAL MODE DURING CYCLE
   54: XIC(CYCLE_IN_PROG)CMP(automaticSeqStep<>0)XIC(manualMode)TON(CYCLE_ALM_TMR[10],?,?);
   55: [XIC(CYCLE_ALM_TMR[10].DN) ,XIC(CYCLE_ALM.12) ]XIO(alarmResetPB)OTE(CYCLE_ALM.12);
   56: XIC(CYCLE_ALM.12)COP(alarmString1[33],alarmStringBuffer,1);
   // X-Axis Motion Alarms
   // =======================================================================================================
   // X-AXIS FAILED TO MOVE HOME
   57: [XIC(TO_DRV1.HOME) ,XIC(X_AXIS_HOME_IN_PROG) ]TON(X_AXIS_ALMTMR[0],?,?);
   58: [XIC(X_AXIS_ALMTMR[0].DN) ,XIC(X_AXIS_HOME_COMPLETE_OSR) XIO(X_AXIS_AT_HOME.Within_Tolerance) ,XIC(X_AXIS_ALARM.0) ]XIO(alarmResetPB)XIO(driveResetHMIPushButton)OTE(X_AXIS_ALARM.0);
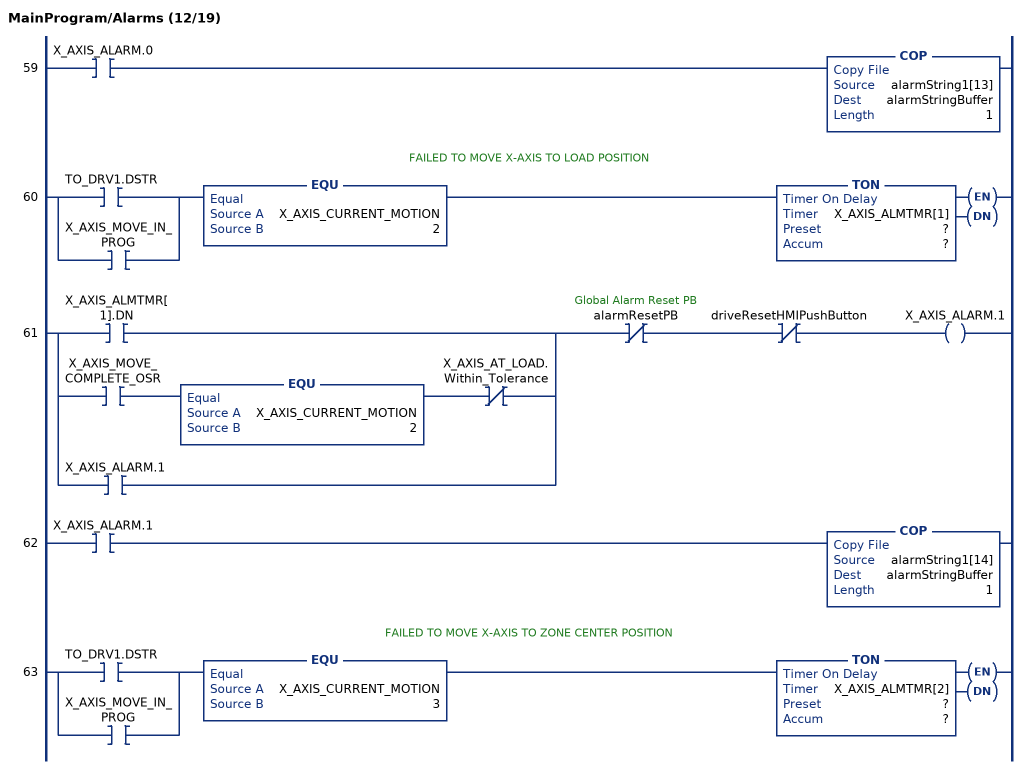
   59: XIC(X_AXIS_ALARM.0)COP(alarmString1[13],alarmStringBuffer,1);
   // FAILED TO MOVE X-AXIS TO LOAD POSITION
   60: [XIC(TO_DRV1.DSTR) ,XIC(X_AXIS_MOVE_IN_PROG) ]EQU(X_AXIS_CURRENT_MOTION,2)TON(X_AXIS_ALMTMR[1],?,?);
   61: [XIC(X_AXIS_ALMTMR[1].DN) ,XIC(X_AXIS_MOVE_COMPLETE_OSR) EQU(X_AXIS_CURRENT_MOTION,2) XIO(X_AXIS_AT_LOAD.Within_Tolerance) ,XIC(X_AXIS_ALARM.1) ]XIO(alarmResetPB)XIO(driveResetHMIPushButton)OTE(X_AXIS_ALARM.1);
   62: XIC(X_AXIS_ALARM.1)COP(alarmString1[14],alarmStringBuffer,1);
   // FAILED TO MOVE X-AXIS TO ZONE CENTER POSITION
   63: [XIC(TO_DRV1.DSTR) ,XIC(X_AXIS_MOVE_IN_PROG) ]EQU(X_AXIS_CURRENT_MOTION,3)TON(X_AXIS_ALMTMR[2],?,?);
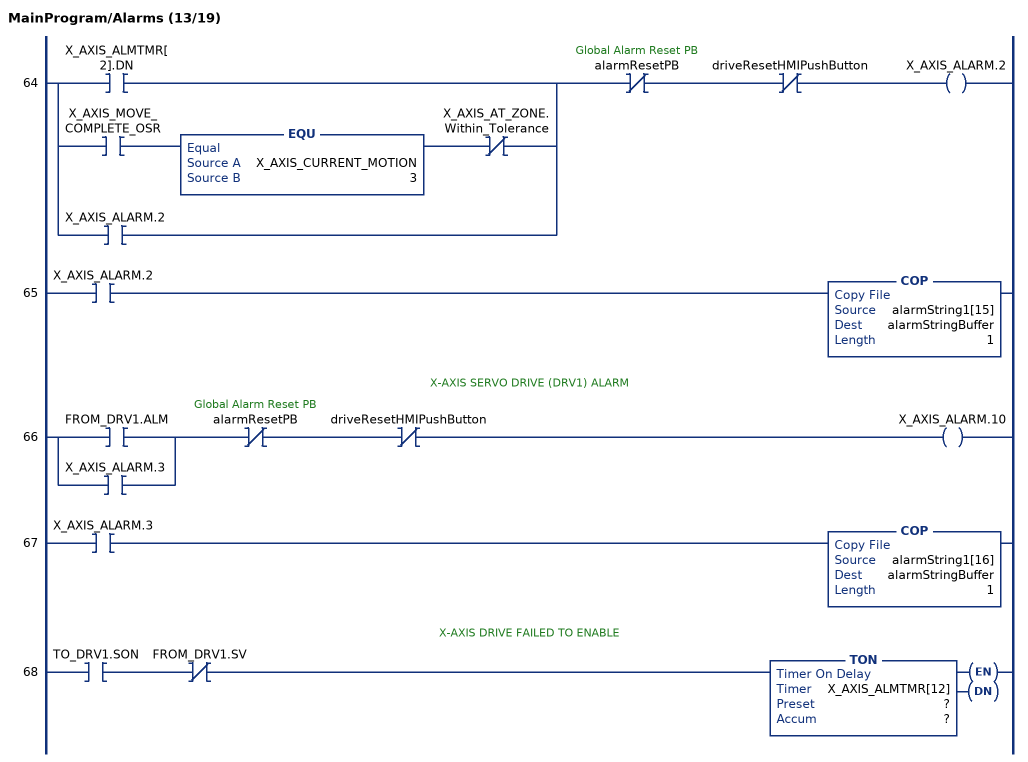
   64: [XIC(X_AXIS_ALMTMR[2].DN) ,XIC(X_AXIS_MOVE_COMPLETE_OSR) EQU(X_AXIS_CURRENT_MOTION,3) XIO(X_AXIS_AT_ZONE.Within_Tolerance) ,XIC(X_AXIS_ALARM.2) ]XIO(alarmResetPB)XIO(driveResetHMIPushButton)OTE(X_AXIS_ALARM.2);
   65: XIC(X_AXIS_ALARM.2)COP(alarmString1[15],alarmStringBuffer,1);
   // X-AXIS SERVO DRIVE (DRV1) ALARM
   66: [XIC(FROM_DRV1.ALM) ,XIC(X_AXIS_ALARM.3) ]XIO(alarmResetPB)XIO(driveResetHMIPushButton)OTE(X_AXIS_ALARM.10);
   67: XIC(X_AXIS_ALARM.3)COP(alarmString1[16],alarmStringBuffer,1);
   // X-AXIS DRIVE FAILED TO ENABLE
   68: XIC(TO_DRV1.SON)XIO(FROM_DRV1.SV)TON(X_AXIS_ALMTMR[12],?,?);
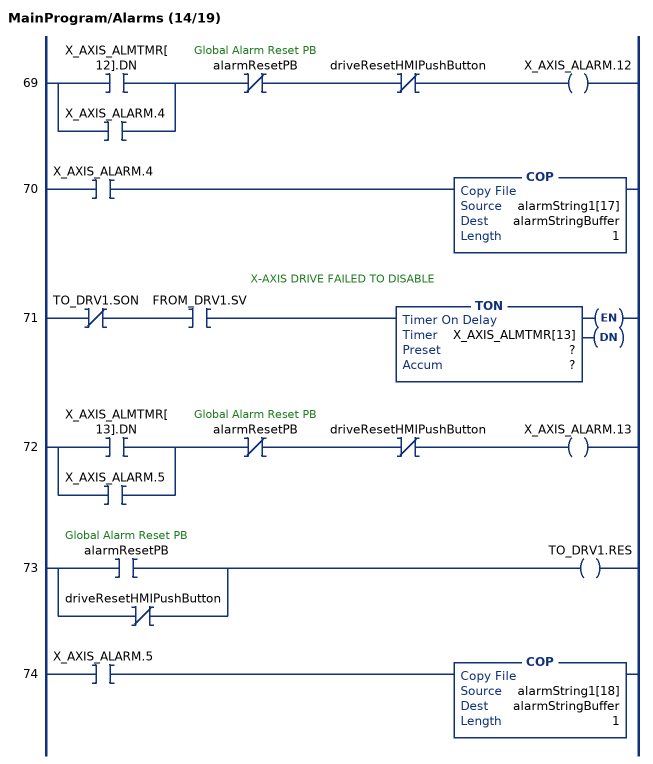
   69: [XIC(X_AXIS_ALMTMR[12].DN) ,XIC(X_AXIS_ALARM.4) ]XIO(alarmResetPB)XIO(driveResetHMIPushButton)OTE(X_AXIS_ALARM.12);
   70: XIC(X_AXIS_ALARM.4)COP(alarmString1[17],alarmStringBuffer,1);
   // X-AXIS DRIVE FAILED TO DISABLE
   71: XIO(TO_DRV1.SON)XIC(FROM_DRV1.SV)TON(X_AXIS_ALMTMR[13],?,?);
   72: [XIC(X_AXIS_ALMTMR[13].DN) ,XIC(X_AXIS_ALARM.5) ]XIO(alarmResetPB)XIO(driveResetHMIPushButton)OTE(X_AXIS_ALARM.13);
   73: [XIC(alarmResetPB) ,XIO(driveResetHMIPushButton) ]OTE(TO_DRV1.RES);
   74: XIC(X_AXIS_ALARM.5)COP(alarmString1[18],alarmStringBuffer,1);
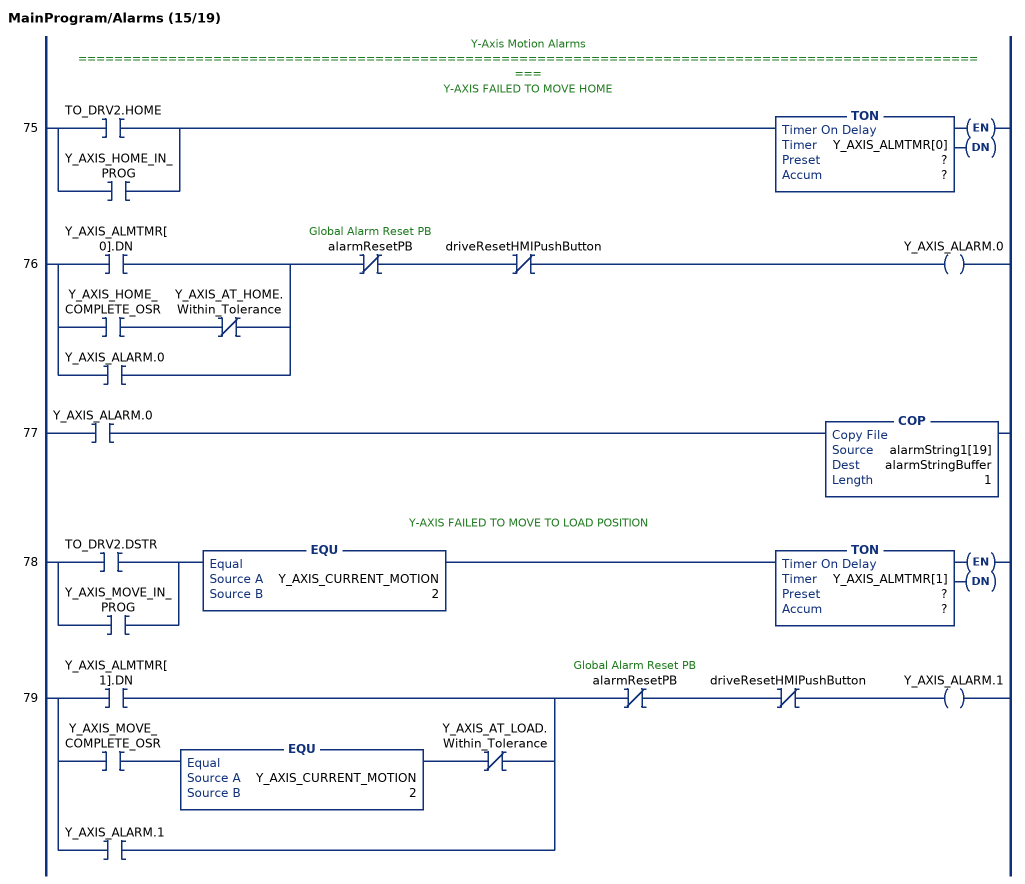
   // Y-Axis Motion Alarms
   // =======================================================================================================
   // Y-AXIS FAILED TO MOVE HOME
   75: [XIC(TO_DRV2.HOME) ,XIC(Y_AXIS_HOME_IN_PROG) ]TON(Y_AXIS_ALMTMR[0],?,?);
   76: [XIC(Y_AXIS_ALMTMR[0].DN) ,XIC(Y_AXIS_HOME_COMPLETE_OSR) XIO(Y_AXIS_AT_HOME.Within_Tolerance) ,XIC(Y_AXIS_ALARM.0) ]XIO(alarmResetPB)XIO(driveResetHMIPushButton)OTE(Y_AXIS_ALARM.0);
   77: XIC(Y_AXIS_ALARM.0)COP(alarmString1[19],alarmStringBuffer,1);
   // Y-AXIS FAILED TO MOVE TO LOAD POSITION
   78: [XIC(TO_DRV2.DSTR) ,XIC(Y_AXIS_MOVE_IN_PROG) ]EQU(Y_AXIS_CURRENT_MOTION,2)TON(Y_AXIS_ALMTMR[1],?,?);
   79: [XIC(Y_AXIS_ALMTMR[1].DN) ,XIC(Y_AXIS_MOVE_COMPLETE_OSR) EQU(Y_AXIS_CURRENT_MOTION,2) XIO(Y_AXIS_AT_LOAD.Within_Tolerance) ,XIC(Y_AXIS_ALARM.1) ]XIO(alarmResetPB)XIO(driveResetHMIPushButton)OTE(Y_AXIS_ALARM.1);
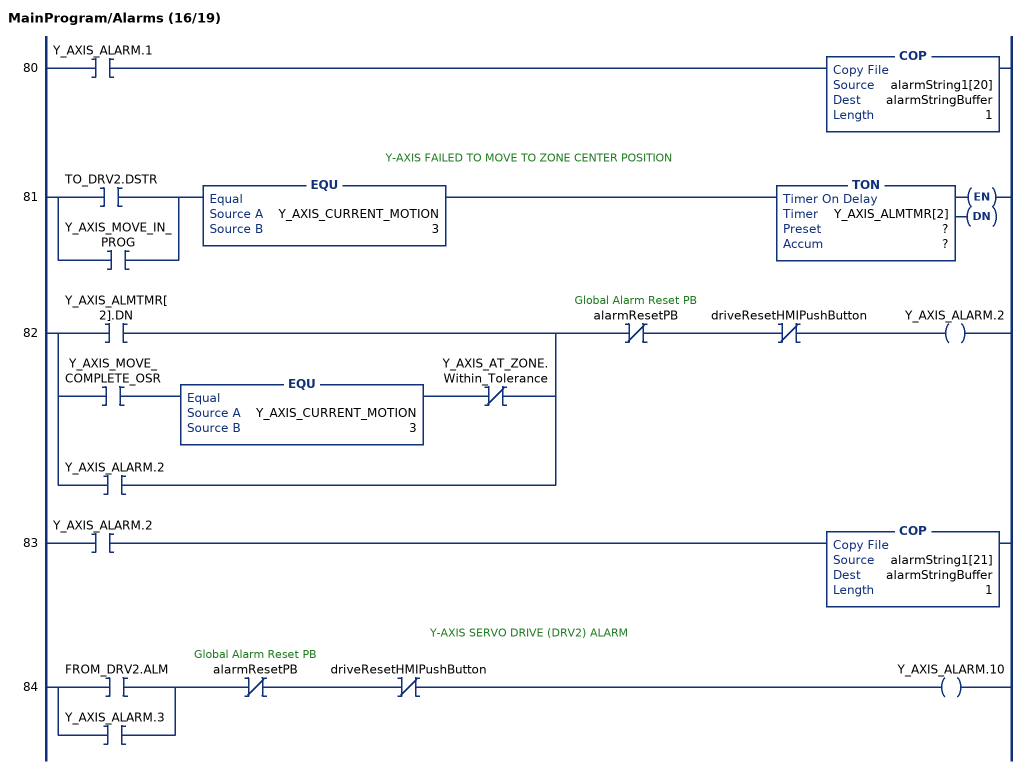
   80: XIC(Y_AXIS_ALARM.1)COP(alarmString1[20],alarmStringBuffer,1);
   // Y-AXIS FAILED TO MOVE TO ZONE CENTER POSITION
   81: [XIC(TO_DRV2.DSTR) ,XIC(Y_AXIS_MOVE_IN_PROG) ]EQU(Y_AXIS_CURRENT_MOTION,3)TON(Y_AXIS_ALMTMR[2],?,?);
   82: [XIC(Y_AXIS_ALMTMR[2].DN) ,XIC(Y_AXIS_MOVE_COMPLETE_OSR) EQU(Y_AXIS_CURRENT_MOTION,3) XIO(Y_AXIS_AT_ZONE.Within_Tolerance) ,XIC(Y_AXIS_ALARM.2) ]XIO(alarmResetPB)XIO(driveResetHMIPushButton)OTE(Y_AXIS_ALARM.2);
   83: XIC(Y_AXIS_ALARM.2)COP(alarmString1[21],alarmStringBuffer,1);
   // Y-AXIS SERVO DRIVE (DRV2) ALARM
   84: [XIC(FROM_DRV2.ALM) ,XIC(Y_AXIS_ALARM.3) ]XIO(alarmResetPB)XIO(driveResetHMIPushButton)OTE(Y_AXIS_ALARM.10);
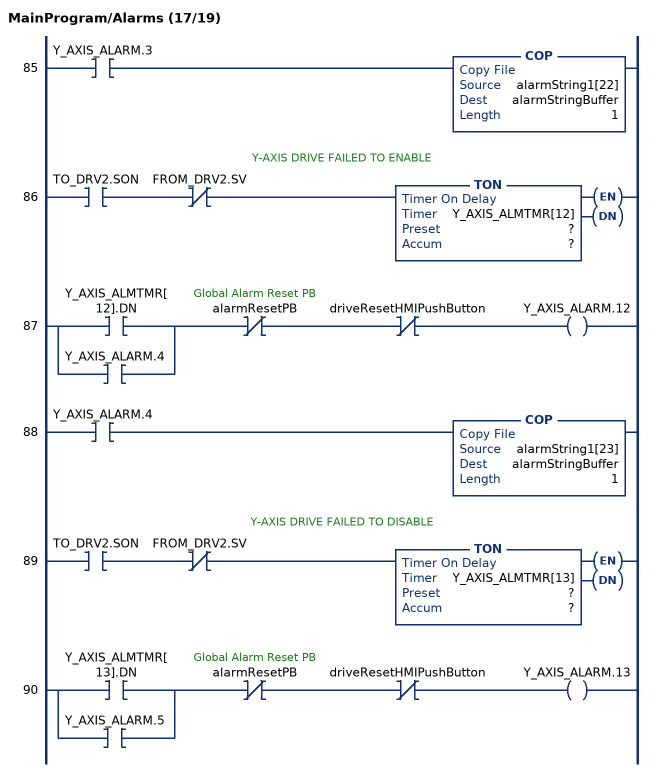
   85: XIC(Y_AXIS_ALARM.3)COP(alarmString1[22],alarmStringBuffer,1);
   // Y-AXIS DRIVE FAILED TO ENABLE
   86: XIC(TO_DRV2.SON)XIO(FROM_DRV2.SV)TON(Y_AXIS_ALMTMR[12],?,?);
   87: [XIC(Y_AXIS_ALMTMR[12].DN) ,XIC(Y_AXIS_ALARM.4) ]XIO(alarmResetPB)XIO(driveResetHMIPushButton)OTE(Y_AXIS_ALARM.12);
   88: XIC(Y_AXIS_ALARM.4)COP(alarmString1[23],alarmStringBuffer,1);
   // Y-AXIS DRIVE FAILED TO DISABLE
   89: XIC(TO_DRV2.SON)XIO(FROM_DRV2.SV)TON(Y_AXIS_ALMTMR[13],?,?);
   90: [XIC(Y_AXIS_ALMTMR[13].DN) ,XIC(Y_AXIS_ALARM.5) ]XIO(alarmResetPB)XIO(driveResetHMIPushButton)OTE(Y_AXIS_ALARM.13);
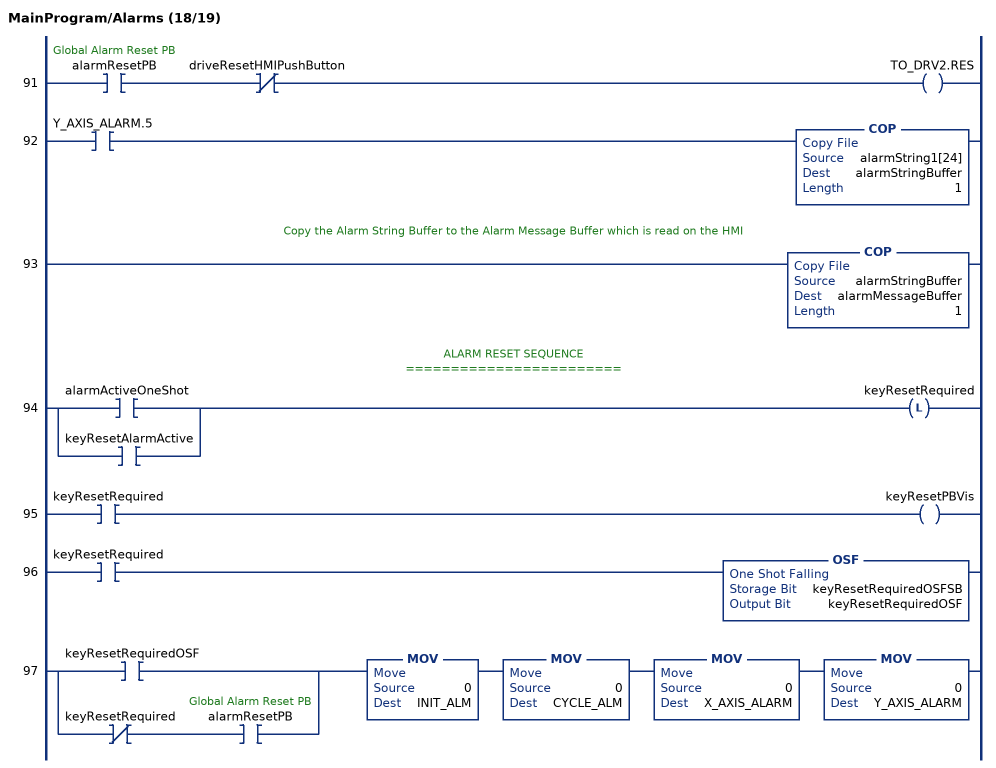
   91: XIC(alarmResetPB)XIO(driveResetHMIPushButton)OTE(TO_DRV2.RES);
   92: XIC(Y_AXIS_ALARM.5)COP(alarmString1[24],alarmStringBuffer,1);
   // Copy the Alarm String Buffer to the Alarm Message Buffer which is read on the HMI
   93: COP(alarmStringBuffer,alarmMessageBuffer,1);
   // ALARM RESET SEQUENCE
   // ========================
   94: [XIC(alarmActiveOneShot) ,XIC(keyResetAlarmActive) ]OTL(keyResetRequired);
   95: XIC(keyResetRequired)OTE(keyResetPBVis);
   96: XIC(keyResetRequired)OSF(keyResetRequiredOSFSB,keyResetRequiredOSF);
   97: [XIC(keyResetRequiredOSF) ,XIO(keyResetRequired) XIC(alarmResetPB) ]MOV(0,INIT_ALM)MOV(0,CYCLE_ALM)MOV(0,X_AXIS_ALARM)MOV(0,Y_AXIS_ALARM);
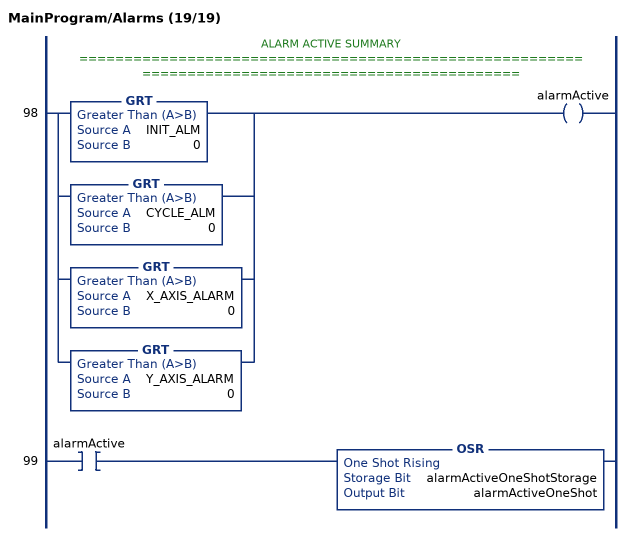
   // ALARM ACTIVE SUMMARY
   // ==================================================================================================
   98: [GRT(INIT_ALM,0) ,GRT(CYCLE_ALM,0) ,GRT(X_AXIS_ALARM,0) ,GRT(Y_AXIS_ALARM,0) ]OTE(alarmActive);
   99: XIC(alarmActive)OSR(alarmActiveOneShotStorage,alarmActiveOneShot);
END_ROUTINE
